FUNCTION_BLOCK Controller_Direction_Speed (* Tamplate for a simple Basic Function Block Type *)
  (* Standard: 61499-2 *)
  (* Version 0.0, 2018-07-24, 4DIAC-IDE, 4DIAC-Consortium *)
  (* Version 1.0, 2016-05-26, AZ, fortiss GmbH *)
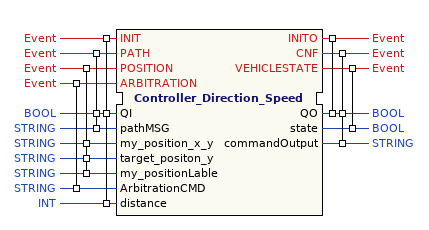
  EVENT_INPUT
    INIT WITH QI, distance; (* Initialization Request *)
    PATH WITH QI, pathMSG;
    POSITION WITH my_position_x_y, target_positon_y, my_positionLable;
    ARBITRATION WITH ArbitrationCMD;
  END_EVENT
  EVENT_OUTPUT
    INITO WITH QO; (* Initialization Confirm *)
    CNF WITH QO, commandOutput; (* Execution Confirmation *)
    VEHICLESTATE WITH state;
  END_EVENT
  VAR_INPUT
    QI : BOOL; (* Input event qualifier *)
    pathMSG : STRING; (* like 1-->3-.... *)
    my_position_x_y : STRING; (* 34_67 *)
    target_positon_y : STRING; (* 54_98 *)
    my_positionLable : STRING; (* e.g.,Piont 3 *)
    ArbitrationCMD : STRING;
    distance : INT;
  END_VAR
  VAR_OUTPUT
    QO : BOOL; (* Output event qualifier *)
    state : BOOL;
    commandOutput : STRING;
  END_VAR
  VAR
    ArbitrateCommand : BOOL := 0; (* Internal Variable *)
    Direction : STRING; (* Internal Variable *)
  END_VAR
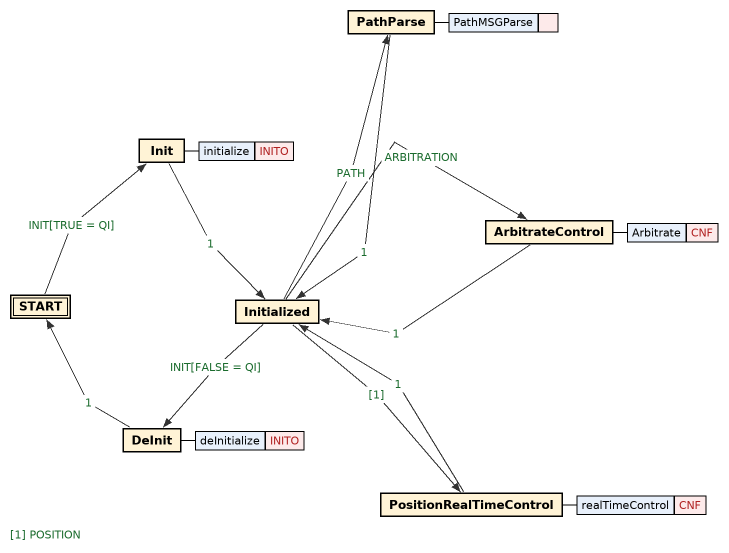
  EC_STATES
    START; (* Initial State *)
    Init : initialize -> INITO; (* Initialization *)
    Initialized;
    DeInit : deInitialize -> INITO;
    PathParse : PathMSGParse;
    ArbitrateControl : Arbitrate -> CNF;
    PositionRealTimeControl : realTimeControl -> CNF;
  END_STATES
  EC_TRANSITIONS
    START TO Init := INIT[TRUE = QI];
    Init TO Initialized := 1;
    DeInit TO START := 1;
    Initialized TO DeInit := INIT[FALSE = QI];
    Initialized TO PathParse := PATH;
    PathParse TO Initialized := 1;
    Initialized TO ArbitrateControl := ARBITRATION;
    ArbitrateControl TO Initialized := 1;
    Initialized TO PositionRealTimeControl := POSITION;
    PositionRealTimeControl TO Initialized := 1;
  END_TRANSITIONS
  ALGORITHM initialize IN ST: (* Initialization algorithm *)
QO := QI;
  END_ALGORITHM
  ALGORITHM deInitialize IN ST: (* Normally executed algorithm *)
QO := FALSE;
  END_ALGORITHM
  ALGORITHM PathMSGParse IN ST: (* new algorithm *)

  END_ALGORITHM
  ALGORITHM Arbitrate IN ST: (* new algorithm *)

  END_ALGORITHM
  ALGORITHM realTimeControl IN ST: (* new algorithm *)

  END_ALGORITHM
END_FUNCTION_BLOCK
